SUBAPPLICATION Uebung_012e_sub_AR (* Numeric Value Input PHYS und Speichern INI mit Subapp (AR Adapter) *)
  (* Standard: 61499-2; Description: Copyright (c) 2026 Meisterschulen am Ostbahnhof This program and the accompanying materials are made available under the terms of the Eclipse Public License 2.0 which is available at https://www.eclipse.org/legal/epl-2.0/ SPDX-License-Identifier: EPL-2.0 *)
  (* Version 1.0, 2026-04-24, Franz Höpfinger, Meisterschulen am Ostbahnhof, AR adapter variant for PHYS REAL INI storage with Subapp *)
  PACKAGE Uebungen;
  IMPORT isobus::UT::Q::const::IDs::ID_NULL;
  IMPORT logiBUS::utils::conversion::phys::NumericObjectPool_S;
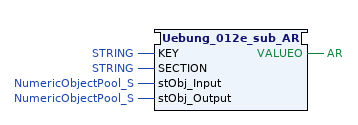
  VAR_INPUT
    KEY : STRING;
    SECTION : STRING;
    stObj_Input : logiBUS::utils::conversion::phys::NumericObjectPool_S := (u16ObjId := ID_NULL, r32Scale := 1.0, i32Offset := 0, u8Decimals := 0);
    stObj_Output : logiBUS::utils::conversion::phys::NumericObjectPool_S := (u16ObjId := ID_NULL, r32Scale := 1.0, i32Offset := 0, u8Decimals := 0);
  END_VAR
  PLUGS
    VALUEO : adapter::types::unidirectional::AR;
  END_PLUGS
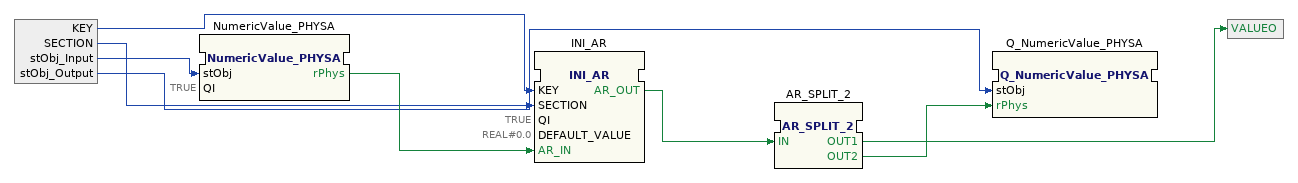
  FBS
    INI_AR : eclipse4diac::storage::INI_AR(QI := TRUE, DEFAULT_VALUE := REAL#0.0);
    NumericValue_PHYSA : isobus::UT::io::NumericValue::NumericValue_PHYSA(QI := TRUE);
    Q_NumericValue_PHYSA : isobus::UT::Q::Q_NumericValue_PHYSA;
    AR_SPLIT_2 : adapter::events::unidirectional::AR_SPLIT_2;
  END_FBS
  DATA_CONNECTIONS
    stObj_Output TO Q_NumericValue_PHYSA.stObj;
    KEY TO INI_AR.KEY;
    SECTION TO INI_AR.SECTION;
    stObj_Input TO NumericValue_PHYSA.stObj;
  END_CONNECTIONS
  ADAPTER_CONNECTIONS
    INI_AR.AR_OUT TO AR_SPLIT_2.IN;
    NumericValue_PHYSA.rPhys TO INI_AR.AR_IN;
    AR_SPLIT_2.OUT1 TO VALUEO;
    AR_SPLIT_2.OUT2 TO Q_NumericValue_PHYSA.rPhys;
  END_CONNECTIONS
END_SUBAPPLICATION
